% RSLogix 500 project binary to gray.RSS, saved by version 8.30.00.16 %
PROJECT "UNTITLED"    % processor: Bul.1763 MicroLogix 1100 Series B %

PROGRAM FILES
  LAD 2   5 rungs

DATA FILES
  O0 OUTPUT  4 elements
  I1 INPUT  6 elements
  S2 STATUS  66 elements
  B3 BINARY  1 elements
  T4 TIMER  1 elements
  C5 COUNTER  1 elements
  R6 CONTROL  1 elements
  N7 INTEGER  1 elements
  F8 FLOAT  1 elements

LADDER 2
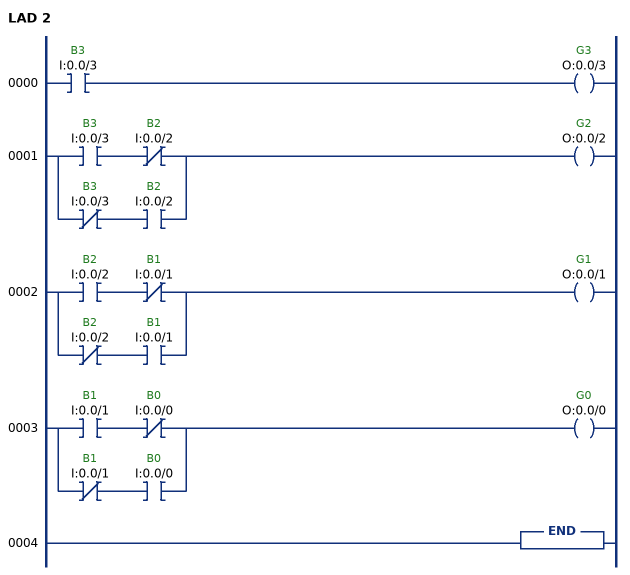
% Rung: 0 %
SOR XIC I:0.0/3 OTE O:0.0/3 EOR
%   I:0.0/3  B3 %
%   O:0.0/3  G3 %
% Rung: 1 %
SOR BST XIC I:0.0/3 XIO I:0.0/2 NXB XIO I:0.0/3 XIC I:0.0/2 BND OTE O:0.0/2 EOR
%   I:0.0/3  B3 %
%   I:0.0/2  B2 %
%   O:0.0/2  G2 %
% Rung: 2 %
SOR BST XIC I:0.0/2 XIO I:0.0/1 NXB XIO I:0.0/2 XIC I:0.0/1 BND OTE O:0.0/1 EOR
%   I:0.0/2  B2 %
%   I:0.0/1  B1 %
%   O:0.0/1  G1 %
% Rung: 3 %
SOR BST XIC I:0.0/1 XIO I:0.0/0 NXB XIO I:0.0/1 XIC I:0.0/0 BND OTE O:0.0/0 EOR
%   I:0.0/1  B1 %
%   I:0.0/0  B0 %
%   O:0.0/0  G0 %
% Rung: 4 %
SOR END EOR
